TYPE DUT_Message :
STRUCT
	Id	: DINT;
	Message	: STRING(255);
END_STRUCT
END_TYPE

(* stored: Version 1.1.0.1, ProductVersion 3.1.4026.18
   DUT DUT_Message: Id {8314dc62-6c29-4c09-a6df-3f7234d2bf3f} *)
